// TIA Portal V17 export
// export: Created 2023-02-14T02:49:47.0513541Z, ExportSetting WithDefaults, DisplayName Totally Integrated Automation Portal, DisplayVersion V17, DisplayName TIA Portal Openness, DisplayVersion V17, DisplayName TIA Portal Teamcenter Gateway, DisplayVersion V17, DisplayName TIA Portal Version Control Interface, DisplayVersion V17, DisplayName SINAMICS Startdrive Advanced, DisplayVersion V17, DisplayName SINAMICS Startdrive G130, G150, S120, S150, SINAMICS MV, S210, DisplayVersion V17, DisplayName SINAMICS Startdrive G110M, G120, G120C, G120D, G120P, G115D, DisplayVersion V17, DisplayName STEP 7 Professional, DisplayVersion V17, DisplayName STEP 7 Safety, DisplayVersion V17, DisplayName WinCC Professional, DisplayVersion V17
FUNCTION_BLOCK "Buffer_Tank"   // FB110, LAD
{ S7_Optimized_Access := 'TRUE' }
VERSION : 0.1
// stored: AutoNumber false, IsIECCheckEnabled false, IsRetainMemResEnabled false, MemoryReserve 100, SetENOAutomatically false, UDAEnableTagReadback false
   VAR_INPUT
      IN_LT01 : Real;
      "Tank w Circulation" : Bool;
      AlarmProd_pasteur : Bool;
      HighLevel_pasteur : Bool;
      IN_FBAV_Inload : Bool;
      IN_FBAV_CIP_Tank : Bool;
      IN_FBAV_CIP_Line : Bool;
      IN_FBAV_Outlet : Bool;
      IN_FBAV_Transfer : Bool;
      IN_FBP_Transfer : Bool;
      IN_FBXA : Bool;
      IN_FBP_Circulation : Bool;
      IN_Product_Ready : Bool;
      IN_Product_TransferOnProg : Bool;
      "Inload Busy" : Bool;
      "CIP Pulse" : Bool;
      "CIP Req OK" : Bool;
      "CIP Supply ON" : Bool;
      "CIP In Progress" : Bool;
      "CIP Complete" : Bool;
      "CIP Busy" : Bool;
   END_VAR
   VAR_OUTPUT
      Out_AV_Inload : Bool;
      Out_AV_Drain_In : Bool;
      Out_AV_CIP_Tank : Bool;
      Out_AV_CIP_Line : Bool;
      Out_AV_Outlet : Bool;
      Out_AV_Transfer : Bool;
      Out_P_Transfer : Bool;
      Out_P_Transfer_SP : Real;
      Out_XA : Bool;
      Out_XA_SP : Real;
      Out_P_Circulation : Bool;
      Out_Prod_Req : Bool;
      Out_Prod_LineOpen : Bool;
      Out_CIP_Tank_Req : Bool;
      Out_CIP_Line_Req : Bool;
      Out_CIP_Tank_LineOpen : Bool;
      Out_CIP_Line_LineOpen : Bool;
   END_VAR
   VAR
      cmd : Struct
         Inload : Bool;
         Drain_In : Bool;
         Ready_for_Transfer : Bool;
         CIP_Tank : Bool;
         CIP_Line : Bool;
         Agitator_Mode : Bool;
         Agitator_Man_OnOff : Bool;
         Agitator_SpeedMode : Bool;
         Circulation : Bool;
      END_STRUCT;
   END_VAR
   VAR RETAIN
      param : Struct
         L_Lo_Lim : Real;
         L_Hi_Lim : Real := 100.0;
         L_Hys : Real := 2.0;
         "Circulation Level" : Real := 20.0;
         SP_Level_HL : Real := 100.0;
         SP_Level_ML : Real := 80.0;
         SP_Level_LL : Real := 10.0;
         DrainIn : DInt := 10;
         SP_Pump_Transfer : Real := 80.0;
         SP_Pump_CIP : Real := 80.0;
         SP_Agitator : Real := 50.0;
         SP_Level_Agi_ON1 : Real := 20.0;
         SP_Level_Agi_OFF1 : Real := 49.0;
         SP_Level_Agi_ON2 : Real := 50.0;
         SP_Level_Agi_OFF2 : Real := 64.0;
         SP_Level_Agi_ON3 : Real := 65.0;
         "CIP Ret On" : Real := 5.0;
         "CIP Ret Off" : Real;
      END_STRUCT;
   END_VAR
   VAR
      state : Struct
         "Tank LL" : Bool;
         "Tank ML" : Bool;
         "Tank HL" : Bool;
         "Tank CIP En" : Bool;
         "Tank CIP" : Bool;
         "Line CIP En" : Bool;
         "Line CIP" : Bool;
         "Ready for Transfer En" : Bool;
         "Ready for Transfer" : Bool;
         Inloading : Bool;
         "Inload En" : Bool;
         L_Agi_ON1 : Bool;
         L_Agi_ON2 : Bool;
         L_Agi_ON3 : Bool;
         Tank_Circulation : Bool;
         "Circulation Enable" : Bool;
         Circulation : Bool;
         "Transfer on Prog" : Bool;
         "CIP Return On" : Bool;
         "CIP Req" : Bool;
      END_STRUCT;
      alwaysOn : Bool;
      L_Hys_Abs : Real;
      Hys_Level_LL : Real;
      Hys_Level_ML : Real;
      Hys_Level_HL : Real;
      Hys_Level_Circ : Real;
   END_VAR
   VAR DB_SPECIFIC
      r : Struct
         PosE1 : Bool;
         PosE2 : Bool;
         PosE3 : Bool;
         PosE4 : Bool;
         PosE5 : Bool;
         PosE6 : Bool;
         PosE7 : Bool;
         PosE8 : Bool;
         PosE9 : Bool;
         PosE10 : Bool;
         PosE11 : Bool;
         PosE12 : Bool;
         PosE13 : Bool;
         PosE14 : Bool;
         PosE15 : Bool;
         PosE16 : Bool;
         PosE17 : Bool;
         PosE18 : Bool;
         PosE19 : Bool;
         PosE20 : Bool;
         PosE21 : Bool;
         PosE22 : Bool;
         PosE23 : Bool;
         PosE24 : Bool;
         PosE25 : Bool;
         PosE26 : Bool;
         PosE27 : Bool;
         PosE28 : Bool;
         PosE29 : Bool;
         PosE30 : Bool;
         PosE31 : Bool;
         PosE32 : Bool;
      END_STRUCT;
      Actuator : Struct
         AV_Inload : Bool;
         AV_Drain_In : Bool;
         AV_Outlet : Bool;
         AV_Transfer : Bool;
         AV_CIP_Tank : Bool;
         AV_CIP_Line : Bool;
         P_Transfer : Bool;
         P_CIP : Bool;
         Agitator_level : Bool;
      END_STRUCT;
   END_VAR
   VAR
      DrainIn_OnTime : TON_TIME;
      DrainIn_OffTime : TOF_TIME;
      InloadAV_OffTime : TOF_TIME;
      DrainIn_MS : DInt;
      L_AgiTim : TON_TIME;
   END_VAR
   VAR_TEMP   // added for the SCL form of the ladder/FBD networks
      _w1 : Bool;
      _w2 : Bool;
      _w3 : Bool;
   END_VAR
BEGIN

REGION Network 1: always On
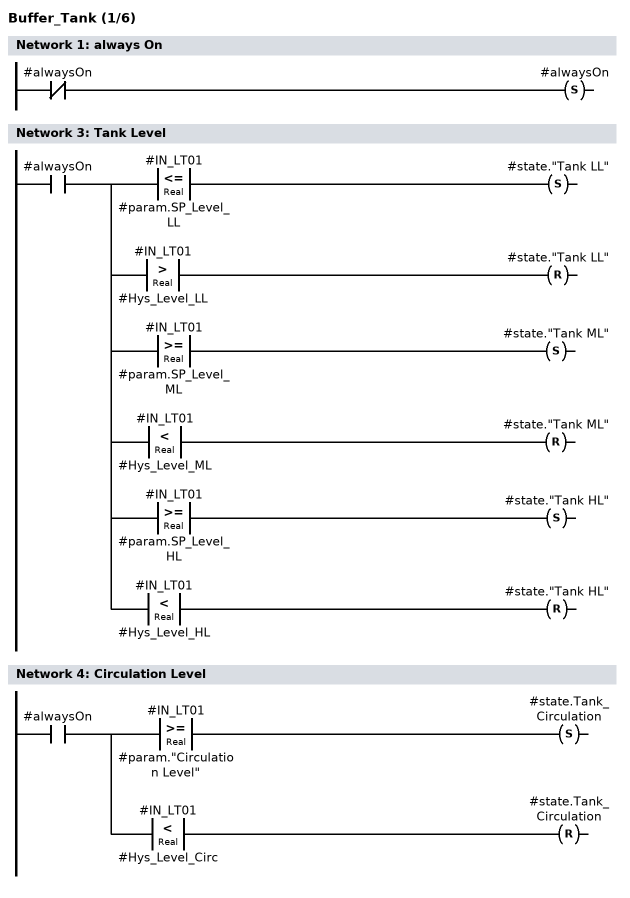
   RUNG wire#powerrail
      I_Contact( #alwaysOn )
      S_Coil( #alwaysOn )
   END_RUNG
   // the same network as SCL:
   IF NOT #alwaysOn THEN #alwaysOn := TRUE; END_IF;
END_REGION

NETWORK
TITLE = Hys Calculation
//Level Hys Absolute
      L     #param.L_Hi_Lim;
      L     #param.L_Lo_Lim;
      -R;
      L     100.0;
      /R;
      L     #param.L_Hys;
      *R;
      T     #L_Hys_Abs;
//Tank High Level
      L     #param.SP_Level_HL;
      L     #L_Hys_Abs;
      -R;
      T     #Hys_Level_HL;
//Tank Mid Level
      L     #param.SP_Level_ML;
      L     #L_Hys_Abs;
      -R;
      T     #Hys_Level_ML;
//Tank Low Level
      L     #param.SP_Level_LL;
      L     #L_Hys_Abs;
      +R;
      T     #Hys_Level_LL;
//Level Circulation
      L     #param."Circulation Level";
      L     #L_Hys_Abs;
      -R;
      T     #Hys_Level_Circ;



REGION Network 3: Tank Level
   RUNG wire#powerrail
      Contact( #alwaysOn )
      wire#w1
      { S7_Templates := "SrcType := Real" } LE_Contact(in1 := #IN_LT01, in2 := #param.SP_Level_LL)
      S_Coil( #state."Tank LL" )
   END_RUNG
   RUNG wire#w1
      { S7_Templates := "SrcType := Real" } GT_Contact(in1 := #IN_LT01, in2 := #Hys_Level_LL)
      R_Coil( #state."Tank LL" )
   END_RUNG
   RUNG wire#w1
      { S7_Templates := "SrcType := Real" } GE_Contact(in1 := #IN_LT01, in2 := #param.SP_Level_ML)
      S_Coil( #state."Tank ML" )
   END_RUNG
   RUNG wire#w1
      { S7_Templates := "SrcType := Real" } LT_Contact(in1 := #IN_LT01, in2 := #Hys_Level_ML)
      R_Coil( #state."Tank ML" )
   END_RUNG
   RUNG wire#w1
      { S7_Templates := "SrcType := Real" } GE_Contact(in1 := #IN_LT01, in2 := #param.SP_Level_HL)
      S_Coil( #state."Tank HL" )
   END_RUNG
   RUNG wire#w1
      { S7_Templates := "SrcType := Real" } LT_Contact(in1 := #IN_LT01, in2 := #Hys_Level_HL)
      R_Coil( #state."Tank HL" )
   END_RUNG
   // the same network as SCL:
   IF #alwaysOn AND (#IN_LT01 <= #param.SP_Level_LL) THEN #state."Tank LL" := TRUE; END_IF;
   IF #alwaysOn AND (#IN_LT01 > #Hys_Level_LL) THEN #state."Tank LL" := FALSE; END_IF;
   IF #alwaysOn AND (#IN_LT01 >= #param.SP_Level_ML) THEN #state."Tank ML" := TRUE; END_IF;
   IF #alwaysOn AND (#IN_LT01 < #Hys_Level_ML) THEN #state."Tank ML" := FALSE; END_IF;
   IF #alwaysOn AND (#IN_LT01 >= #param.SP_Level_HL) THEN #state."Tank HL" := TRUE; END_IF;
   IF #alwaysOn AND (#IN_LT01 < #Hys_Level_HL) THEN #state."Tank HL" := FALSE; END_IF;
END_REGION

REGION Network 4: Circulation Level
   RUNG wire#powerrail
      Contact( #alwaysOn )
      wire#w1
      { S7_Templates := "SrcType := Real" } GE_Contact(in1 := #IN_LT01, in2 := #param."Circulation Level")
      S_Coil( #state.Tank_Circulation )
   END_RUNG
   RUNG wire#w1
      { S7_Templates := "SrcType := Real" } LT_Contact(in1 := #IN_LT01, in2 := #Hys_Level_Circ)
      R_Coil( #state.Tank_Circulation )
   END_RUNG
   // the same network as SCL:
   IF #alwaysOn AND (#IN_LT01 >= #param."Circulation Level") THEN #state.Tank_Circulation := TRUE; END_IF;
   IF #alwaysOn AND (#IN_LT01 < #Hys_Level_Circ) THEN #state.Tank_Circulation := FALSE; END_IF;
END_REGION

REGION Network 5: Agitator Level ON-OFF
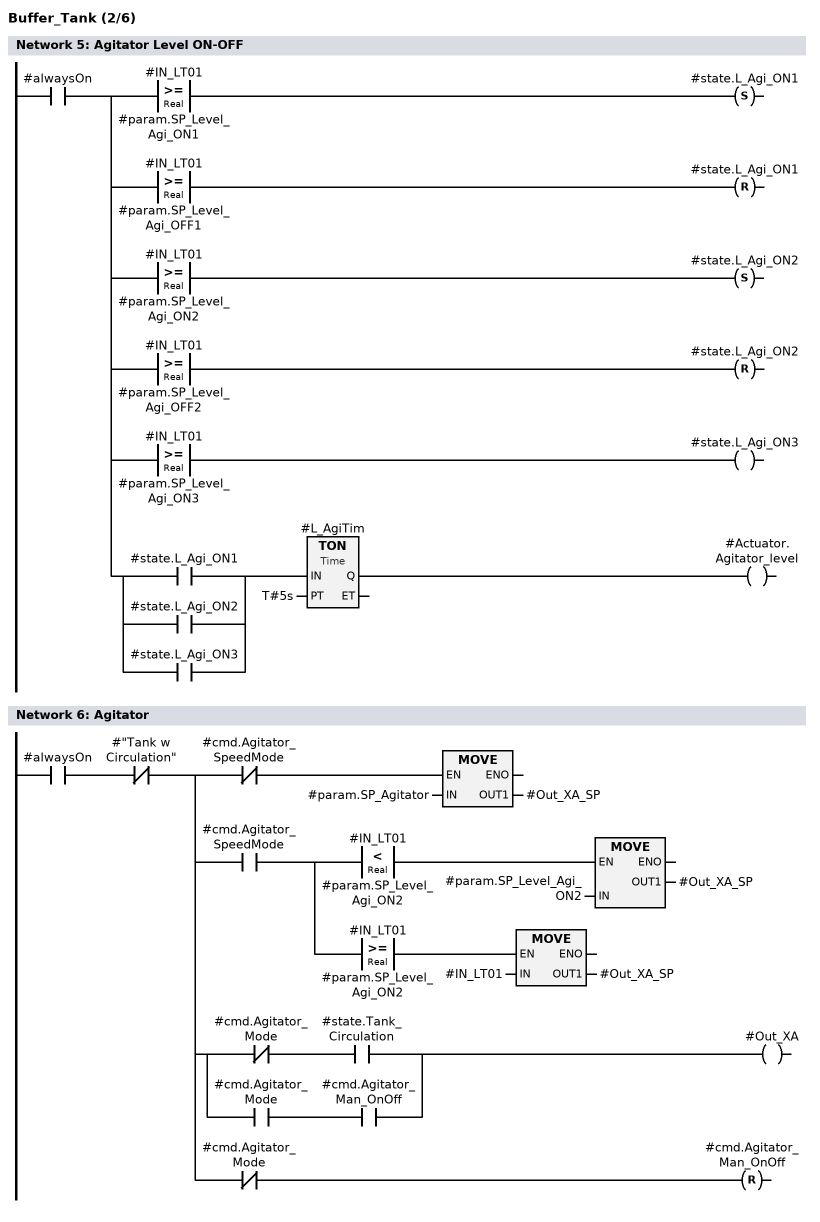
   RUNG wire#powerrail
      Contact( #alwaysOn )
      wire#w1
      { S7_Templates := "SrcType := Real" } GE_Contact(in1 := #IN_LT01, in2 := #param.SP_Level_Agi_ON1)
      S_Coil( #state.L_Agi_ON1 )
   END_RUNG
   RUNG wire#w1
      { S7_Templates := "SrcType := Real" } GE_Contact(in1 := #IN_LT01, in2 := #param.SP_Level_Agi_OFF1)
      R_Coil( #state.L_Agi_ON1 )
   END_RUNG
   RUNG wire#w1
      { S7_Templates := "SrcType := Real" } GE_Contact(in1 := #IN_LT01, in2 := #param.SP_Level_Agi_ON2)
      S_Coil( #state.L_Agi_ON2 )
   END_RUNG
   RUNG wire#w1
      { S7_Templates := "SrcType := Real" } GE_Contact(in1 := #IN_LT01, in2 := #param.SP_Level_Agi_OFF2)
      R_Coil( #state.L_Agi_ON2 )
   END_RUNG
   RUNG wire#w1
      { S7_Templates := "SrcType := Real" } GE_Contact(in1 := #IN_LT01, in2 := #param.SP_Level_Agi_ON3)
      Coil( #state.L_Agi_ON3 )
   END_RUNG
   RUNG wire#w1
      Contact( #state.L_Agi_ON1 )
      wire#w2
      { S7_Templates := "time_type := Time" } #L_AgiTim.TON(pt := T#5s, et =>)
      Coil( #Actuator.Agitator_level )
   END_RUNG
   RUNG wire#w1
      Contact( #state.L_Agi_ON2 )
   END_RUNG wire#w2
   RUNG wire#w1
      Contact( #state.L_Agi_ON3 )
   END_RUNG wire#w2
   // the same network as SCL:
   IF #alwaysOn AND (#IN_LT01 >= #param.SP_Level_Agi_ON1) THEN #state.L_Agi_ON1 := TRUE; END_IF;
   IF #alwaysOn AND (#IN_LT01 >= #param.SP_Level_Agi_OFF1) THEN #state.L_Agi_ON1 := FALSE; END_IF;
   IF #alwaysOn AND (#IN_LT01 >= #param.SP_Level_Agi_ON2) THEN #state.L_Agi_ON2 := TRUE; END_IF;
   IF #alwaysOn AND (#IN_LT01 >= #param.SP_Level_Agi_OFF2) THEN #state.L_Agi_ON2 := FALSE; END_IF;
   #state.L_Agi_ON3 := #alwaysOn AND (#IN_LT01 >= #param.SP_Level_Agi_ON3);
   #L_AgiTim(IN := #alwaysOn AND (#state.L_Agi_ON1 OR #state.L_Agi_ON2 OR #state.L_Agi_ON3), PT := T#5s);   // TON
   #Actuator.Agitator_level := #L_AgiTim.Q;
END_REGION

REGION Network 6: Agitator
   RUNG wire#powerrail
      Contact( #alwaysOn )
      I_Contact( #"Tank w Circulation" )
      wire#w1
      I_Contact( #cmd.Agitator_SpeedMode )
      Move(in := #param.SP_Agitator, out1 => #Out_XA_SP)
   END_RUNG
   RUNG wire#w1
      Contact( #cmd.Agitator_SpeedMode )
      wire#w2
      { S7_Templates := "SrcType := Real" } LT_Contact(in1 := #IN_LT01, in2 := #param.SP_Level_Agi_ON2)
      Move(in := #param.SP_Level_Agi_ON2, out1 => #Out_XA_SP)
   END_RUNG
   RUNG wire#w2
      { S7_Templates := "SrcType := Real" } GE_Contact(in1 := #IN_LT01, in2 := #param.SP_Level_Agi_ON2)
      Move(in := #IN_LT01, out1 => #Out_XA_SP)
   END_RUNG
   RUNG wire#w1
      I_Contact( #cmd.Agitator_Mode )
      Contact( #state.Tank_Circulation )
      wire#w3
      Coil( #Out_XA )
   END_RUNG
   RUNG wire#w1
      Contact( #cmd.Agitator_Mode )
      Contact( #cmd.Agitator_Man_OnOff )
   END_RUNG wire#w3
   RUNG wire#w1
      I_Contact( #cmd.Agitator_Mode )
      R_Coil( #cmd.Agitator_Man_OnOff )
   END_RUNG
   // the same network as SCL:
   #_w1 := #alwaysOn AND NOT #"Tank w Circulation";
   IF #_w1 AND NOT #cmd.Agitator_SpeedMode THEN #Out_XA_SP := #param.SP_Agitator; END_IF;
   #_w2 := #_w1 AND #cmd.Agitator_SpeedMode;
   IF #_w2 AND (#IN_LT01 < #param.SP_Level_Agi_ON2) THEN #Out_XA_SP := #param.SP_Level_Agi_ON2; END_IF;
   IF #_w2 AND (#IN_LT01 >= #param.SP_Level_Agi_ON2) THEN #Out_XA_SP := #IN_LT01; END_IF;
   #Out_XA := #_w1 AND ((NOT #cmd.Agitator_Mode AND #state.Tank_Circulation) OR (#cmd.Agitator_Mode AND #cmd.Agitator_Man_OnOff));
   IF #_w1 AND NOT #cmd.Agitator_Mode THEN #cmd.Agitator_Man_OnOff := FALSE; END_IF;
END_REGION

REGION Network 7: Circulation
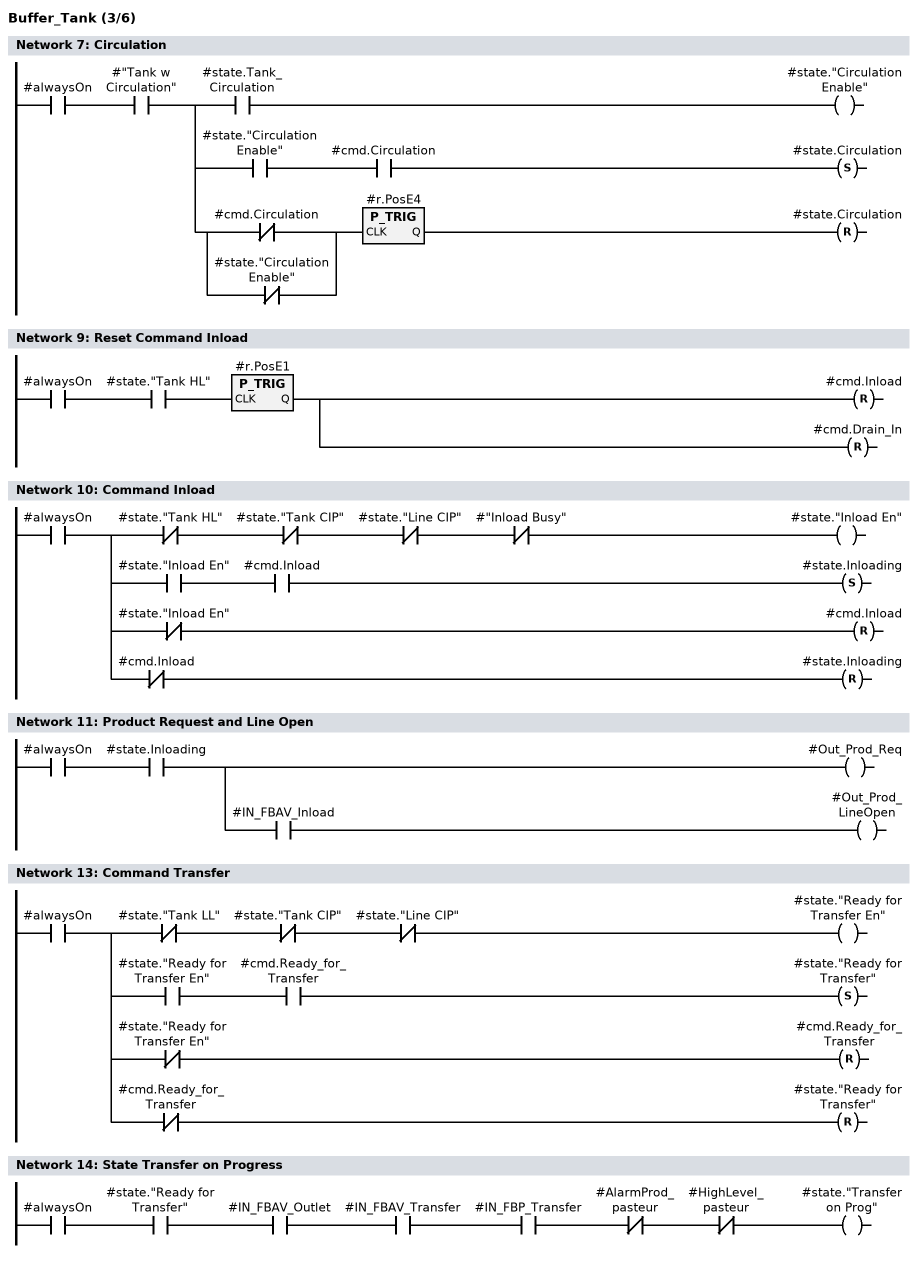
   RUNG wire#powerrail
      Contact( #alwaysOn )
      Contact( #"Tank w Circulation" )
      wire#w1
      Contact( #state.Tank_Circulation )
      Coil( #state."Circulation Enable" )
   END_RUNG
   RUNG wire#w1
      Contact( #state."Circulation Enable" )
      Contact( #cmd.Circulation )
      S_Coil( #state.Circulation )
   END_RUNG
   RUNG wire#w1
      I_Contact( #cmd.Circulation )
      wire#w2
      P_Trig( #r.PosE4 )
      R_Coil( #state.Circulation )
   END_RUNG
   RUNG wire#w1
      I_Contact( #state."Circulation Enable" )
   END_RUNG wire#w2
   // the same network as SCL:
   #_w1 := #alwaysOn AND #"Tank w Circulation";
   #state."Circulation Enable" := #_w1 AND #state.Tank_Circulation;
   IF #_w1 AND #state."Circulation Enable" AND #cmd.Circulation THEN #state.Circulation := TRUE; END_IF;
   #_w2 := #_w1 AND (NOT #cmd.Circulation OR NOT #state."Circulation Enable");
   #_w3 := #_w2 AND NOT #r.PosE4;   // rising edge
   #r.PosE4 := #_w2;
   IF #_w3 THEN #state.Circulation := FALSE; END_IF;
END_REGION

REGION Network 9: Reset Command Inload
   RUNG wire#powerrail
      Contact( #alwaysOn )
      Contact( #state."Tank HL" )
      P_Trig( #r.PosE1 )
      wire#w1
      R_Coil( #cmd.Inload )
   END_RUNG
   RUNG wire#w1
      R_Coil( #cmd.Drain_In )
   END_RUNG
   // the same network as SCL:
   #_w1 := #alwaysOn AND #state."Tank HL";
   #_w2 := #_w1 AND NOT #r.PosE1;   // rising edge
   #r.PosE1 := #_w1;
   IF #_w2 THEN
       #cmd.Inload := FALSE;
       #cmd.Drain_In := FALSE;
   END_IF;
END_REGION

REGION Network 10: Command Inload
   RUNG wire#powerrail
      Contact( #alwaysOn )
      wire#w1
      I_Contact( #state."Tank HL" )
      I_Contact( #state."Tank CIP" )
      I_Contact( #state."Line CIP" )
      I_Contact( #"Inload Busy" )
      Coil( #state."Inload En" )
   END_RUNG
   RUNG wire#w1
      Contact( #state."Inload En" )
      Contact( #cmd.Inload )
      S_Coil( #state.Inloading )
   END_RUNG
   RUNG wire#w1
      I_Contact( #state."Inload En" )
      R_Coil( #cmd.Inload )
   END_RUNG
   RUNG wire#w1
      I_Contact( #cmd.Inload )
      R_Coil( #state.Inloading )
   END_RUNG
   // the same network as SCL:
   #state."Inload En" := #alwaysOn AND NOT #state."Tank HL" AND NOT #state."Tank CIP" AND NOT #state."Line CIP" AND NOT #"Inload Busy";
   IF #alwaysOn AND #state."Inload En" AND #cmd.Inload THEN #state.Inloading := TRUE; END_IF;
   IF #alwaysOn AND NOT #state."Inload En" THEN #cmd.Inload := FALSE; END_IF;
   IF #alwaysOn AND NOT #cmd.Inload THEN #state.Inloading := FALSE; END_IF;
END_REGION

REGION Network 11: Product Request and Line Open
   RUNG wire#powerrail
      Contact( #alwaysOn )
      Contact( #state.Inloading )
      wire#w1
      Coil( #Out_Prod_Req )
   END_RUNG
   RUNG wire#w1
      Contact( #IN_FBAV_Inload )
      Coil( #Out_Prod_LineOpen )
   END_RUNG
   // the same network as SCL:
   #Out_Prod_Req := #alwaysOn AND #state.Inloading;
   #Out_Prod_LineOpen := #Out_Prod_Req AND #IN_FBAV_Inload;
END_REGION

REGION Network 13: Command Transfer
   RUNG wire#powerrail
      Contact( #alwaysOn )
      wire#w1
      I_Contact( #state."Tank LL" )
      I_Contact( #state."Tank CIP" )
      I_Contact( #state."Line CIP" )
      Coil( #state."Ready for Transfer En" )
   END_RUNG
   RUNG wire#w1
      Contact( #state."Ready for Transfer En" )
      Contact( #cmd.Ready_for_Transfer )
      S_Coil( #state."Ready for Transfer" )
   END_RUNG
   RUNG wire#w1
      I_Contact( #state."Ready for Transfer En" )
      R_Coil( #cmd.Ready_for_Transfer )
   END_RUNG
   RUNG wire#w1
      I_Contact( #cmd.Ready_for_Transfer )
      R_Coil( #state."Ready for Transfer" )
   END_RUNG
   // the same network as SCL:
   #state."Ready for Transfer En" := #alwaysOn AND NOT #state."Tank LL" AND NOT #state."Tank CIP" AND NOT #state."Line CIP";
   IF #alwaysOn AND #state."Ready for Transfer En" AND #cmd.Ready_for_Transfer THEN
       #state."Ready for Transfer" := TRUE;
   END_IF;
   IF #alwaysOn AND NOT #state."Ready for Transfer En" THEN #cmd.Ready_for_Transfer := FALSE; END_IF;
   IF #alwaysOn AND NOT #cmd.Ready_for_Transfer THEN #state."Ready for Transfer" := FALSE; END_IF;
END_REGION

REGION Network 14: State Transfer on Progress
   RUNG wire#powerrail
      Contact( #alwaysOn )
      Contact( #state."Ready for Transfer" )
      Contact( #IN_FBAV_Outlet )
      Contact( #IN_FBAV_Transfer )
      Contact( #IN_FBP_Transfer )
      I_Contact( #AlarmProd_pasteur )
      I_Contact( #HighLevel_pasteur )
      Coil( #state."Transfer on Prog" )
   END_RUNG
   // the same network as SCL:
   #state."Transfer on Prog" := #alwaysOn AND #state."Ready for Transfer" AND #IN_FBAV_Outlet AND #IN_FBAV_Transfer AND #IN_FBP_Transfer AND NOT #AlarmProd_pasteur AND NOT #HighLevel_pasteur;
END_REGION

REGION Network 16: Command CIP
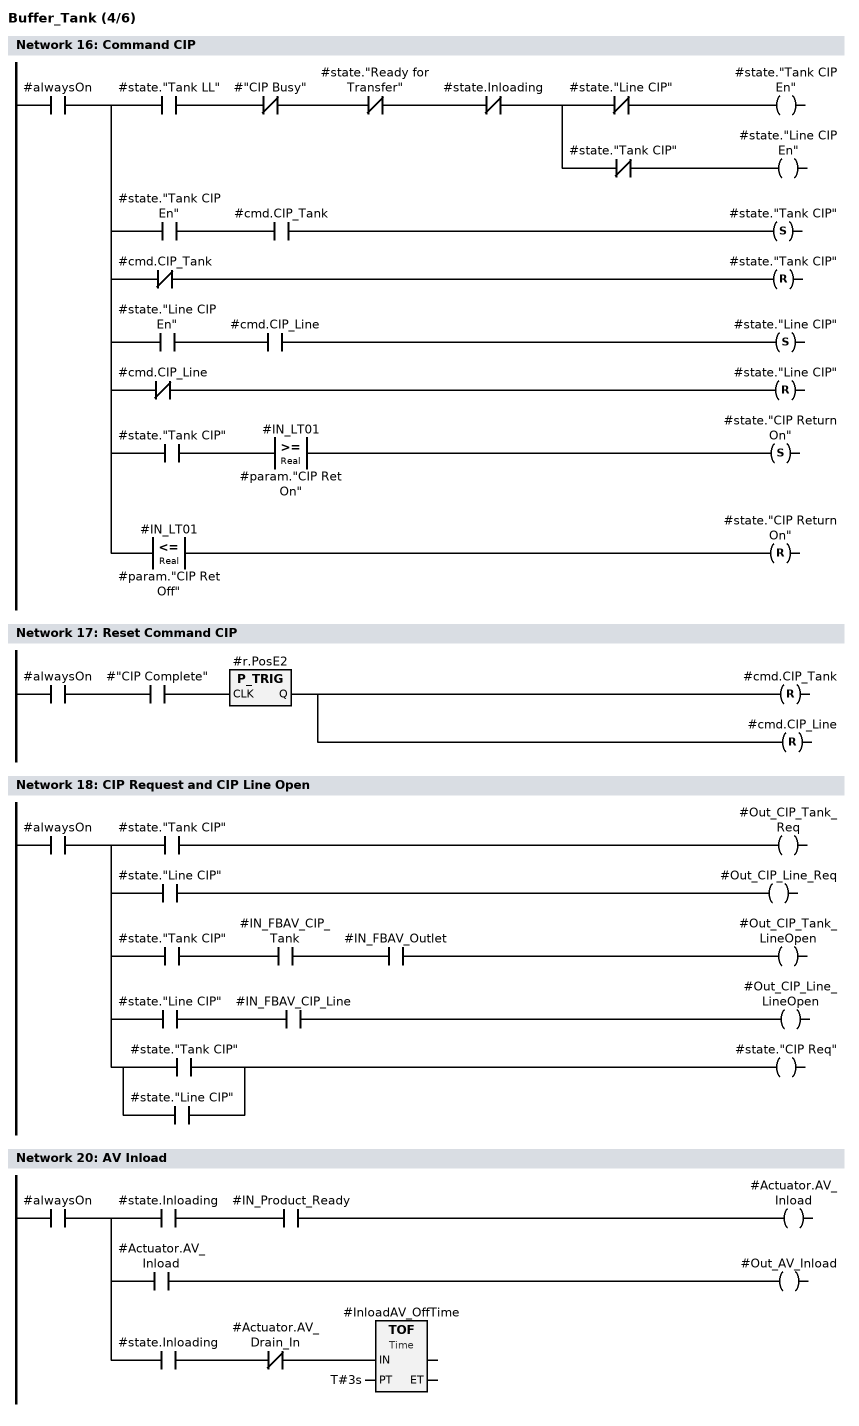
   RUNG wire#powerrail
      Contact( #alwaysOn )
      wire#w1
      Contact( #state."Tank LL" )
      I_Contact( #"CIP Busy" )
      I_Contact( #state."Ready for Transfer" )
      I_Contact( #state.Inloading )
      wire#w2
      I_Contact( #state."Line CIP" )
      Coil( #state."Tank CIP En" )
   END_RUNG
   RUNG wire#w2
      I_Contact( #state."Tank CIP" )
      Coil( #state."Line CIP En" )
   END_RUNG
   RUNG wire#w1
      Contact( #state."Tank CIP En" )
      Contact( #cmd.CIP_Tank )
      S_Coil( #state."Tank CIP" )
   END_RUNG
   RUNG wire#w1
      I_Contact( #cmd.CIP_Tank )
      R_Coil( #state."Tank CIP" )
   END_RUNG
   RUNG wire#w1
      Contact( #state."Line CIP En" )
      Contact( #cmd.CIP_Line )
      S_Coil( #state."Line CIP" )
   END_RUNG
   RUNG wire#w1
      I_Contact( #cmd.CIP_Line )
      R_Coil( #state."Line CIP" )
   END_RUNG
   RUNG wire#w1
      Contact( #state."Tank CIP" )
      { S7_Templates := "SrcType := Real" } GE_Contact(in1 := #IN_LT01, in2 := #param."CIP Ret On")
      S_Coil( #state."CIP Return On" )
   END_RUNG
   RUNG wire#w1
      { S7_Templates := "SrcType := Real" } LE_Contact(in1 := #IN_LT01, in2 := #param."CIP Ret Off")
      R_Coil( #state."CIP Return On" )
   END_RUNG
   // the same network as SCL:
   #_w1 := #alwaysOn AND #state."Tank LL" AND NOT #"CIP Busy" AND NOT #state."Ready for Transfer" AND NOT #state.Inloading;
   #state."Tank CIP En" := #_w1 AND NOT #state."Line CIP";
   #state."Line CIP En" := #_w1 AND NOT #state."Tank CIP";
   IF #alwaysOn AND #state."Tank CIP En" AND #cmd.CIP_Tank THEN #state."Tank CIP" := TRUE; END_IF;
   IF #alwaysOn AND NOT #cmd.CIP_Tank THEN #state."Tank CIP" := FALSE; END_IF;
   IF #alwaysOn AND #state."Line CIP En" AND #cmd.CIP_Line THEN #state."Line CIP" := TRUE; END_IF;
   IF #alwaysOn AND NOT #cmd.CIP_Line THEN #state."Line CIP" := FALSE; END_IF;
   IF #alwaysOn AND #state."Tank CIP" AND (#IN_LT01 >= #param."CIP Ret On") THEN
       #state."CIP Return On" := TRUE;
   END_IF;
   IF #alwaysOn AND (#IN_LT01 <= #param."CIP Ret Off") THEN #state."CIP Return On" := FALSE; END_IF;
END_REGION

REGION Network 17: Reset Command CIP
   RUNG wire#powerrail
      Contact( #alwaysOn )
      Contact( #"CIP Complete" )
      P_Trig( #r.PosE2 )
      wire#w1
      R_Coil( #cmd.CIP_Tank )
   END_RUNG
   RUNG wire#w1
      R_Coil( #cmd.CIP_Line )
   END_RUNG
   // the same network as SCL:
   #_w1 := #alwaysOn AND #"CIP Complete";
   #_w2 := #_w1 AND NOT #r.PosE2;   // rising edge
   #r.PosE2 := #_w1;
   IF #_w2 THEN
       #cmd.CIP_Tank := FALSE;
       #cmd.CIP_Line := FALSE;
   END_IF;
END_REGION

REGION Network 18: CIP Request and CIP Line Open
   RUNG wire#powerrail
      Contact( #alwaysOn )
      wire#w1
      Contact( #state."Tank CIP" )
      Coil( #Out_CIP_Tank_Req )
   END_RUNG
   RUNG wire#w1
      Contact( #state."Line CIP" )
      Coil( #Out_CIP_Line_Req )
   END_RUNG
   RUNG wire#w1
      Contact( #state."Tank CIP" )
      Contact( #IN_FBAV_CIP_Tank )
      Contact( #IN_FBAV_Outlet )
      Coil( #Out_CIP_Tank_LineOpen )
   END_RUNG
   RUNG wire#w1
      Contact( #state."Line CIP" )
      Contact( #IN_FBAV_CIP_Line )
      Coil( #Out_CIP_Line_LineOpen )
   END_RUNG
   RUNG wire#w1
      Contact( #state."Tank CIP" )
      wire#w2
      Coil( #state."CIP Req" )
   END_RUNG
   RUNG wire#w1
      Contact( #state."Line CIP" )
   END_RUNG wire#w2
   // the same network as SCL:
   #Out_CIP_Tank_Req := #alwaysOn AND #state."Tank CIP";
   #Out_CIP_Line_Req := #alwaysOn AND #state."Line CIP";
   #Out_CIP_Tank_LineOpen := #alwaysOn AND #state."Tank CIP" AND #IN_FBAV_CIP_Tank AND #IN_FBAV_Outlet;
   #Out_CIP_Line_LineOpen := #alwaysOn AND #state."Line CIP" AND #IN_FBAV_CIP_Line;
   #state."CIP Req" := #alwaysOn AND (#state."Tank CIP" OR #state."Line CIP");
END_REGION

REGION Network 20: AV Inload
   RUNG wire#powerrail
      Contact( #alwaysOn )
      wire#w1
      Contact( #state.Inloading )
      Contact( #IN_Product_Ready )
      Coil( #Actuator.AV_Inload )
   END_RUNG
   RUNG wire#w1
      Contact( #Actuator.AV_Inload )
      Coil( #Out_AV_Inload )
   END_RUNG
   RUNG wire#w1
      Contact( #state.Inloading )
      I_Contact( #Actuator.AV_Drain_In )
      { S7_Templates := "time_type := Time" } #InloadAV_OffTime.TOF(pt := T#3s, et =>)
   END_RUNG
   // the same network as SCL:
   #Actuator.AV_Inload := #alwaysOn AND #state.Inloading AND #IN_Product_Ready;
   #Out_AV_Inload := #alwaysOn AND #Actuator.AV_Inload;
   #InloadAV_OffTime(IN := #alwaysOn AND #state.Inloading AND NOT #Actuator.AV_Drain_In, PT := T#3s);   // TOF
END_REGION

REGION Network 21: AV Drain In
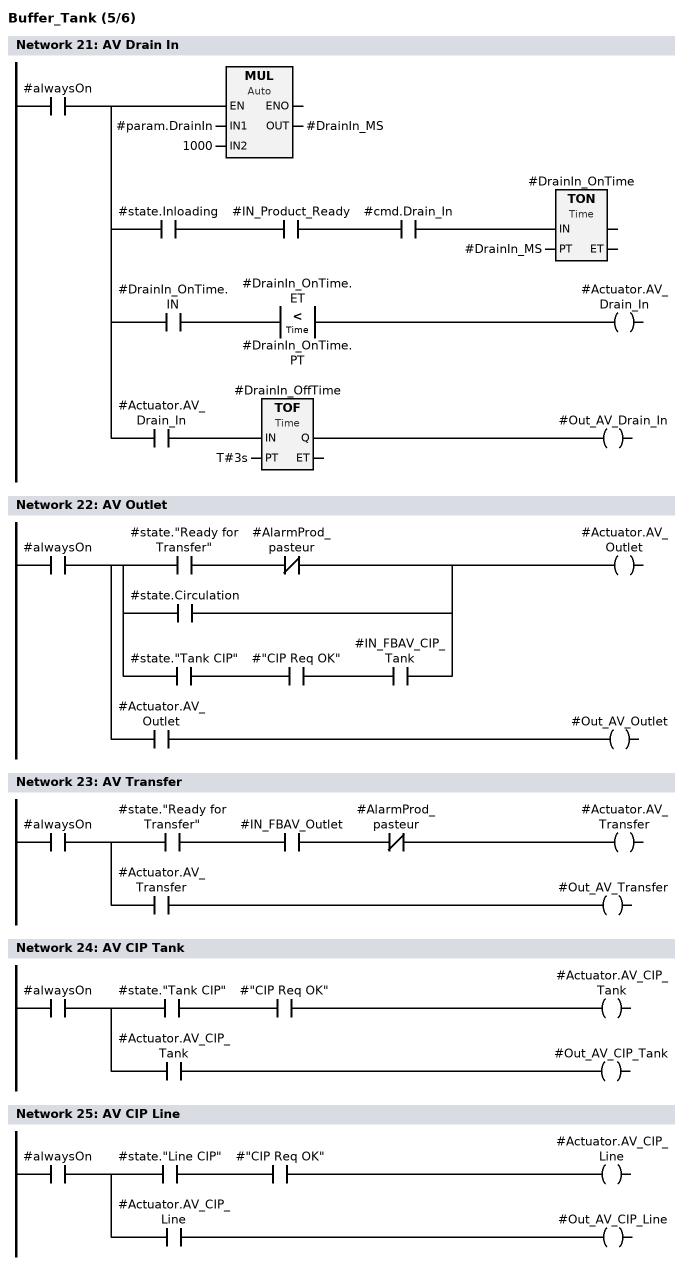
   RUNG wire#powerrail
      Contact( #alwaysOn )
      wire#w1
      Mul(in1 := #param.DrainIn, in2 := 1000, out => #DrainIn_MS)
   END_RUNG
   RUNG wire#w1
      Contact( #state.Inloading )
      Contact( #IN_Product_Ready )
      Contact( #cmd.Drain_In )
      { S7_Templates := "time_type := Time" } #DrainIn_OnTime.TON(pt := #DrainIn_MS, et =>)
   END_RUNG
   RUNG wire#w1
      Contact( #DrainIn_OnTime.IN )
      { S7_Templates := "SrcType := Time" } LT_Contact(in1 := #DrainIn_OnTime.ET, in2 := #DrainIn_OnTime.PT)
      Coil( #Actuator.AV_Drain_In )
   END_RUNG
   RUNG wire#w1
      Contact( #Actuator.AV_Drain_In )
      { S7_Templates := "time_type := Time" } #DrainIn_OffTime.TOF(pt := T#3s, et =>)
      Coil( #Out_AV_Drain_In )
   END_RUNG
   // the same network as SCL:
   IF #alwaysOn THEN #DrainIn_MS := #param.DrainIn * 1000; END_IF;
   #DrainIn_OnTime(IN := #alwaysOn AND #state.Inloading AND #IN_Product_Ready AND #cmd.Drain_In,   // TON
                   PT := #DrainIn_MS);
   #Actuator.AV_Drain_In := #alwaysOn AND #DrainIn_OnTime.IN AND (#DrainIn_OnTime.ET < #DrainIn_OnTime.PT);
   #DrainIn_OffTime(IN := #alwaysOn AND #Actuator.AV_Drain_In, PT := T#3s);   // TOF
   #Out_AV_Drain_In := #DrainIn_OffTime.Q;
END_REGION

REGION Network 22: AV Outlet
   RUNG wire#powerrail
      Contact( #alwaysOn )
      wire#w1
      Contact( #state."Ready for Transfer" )
      I_Contact( #AlarmProd_pasteur )
      wire#w2
      Coil( #Actuator.AV_Outlet )
   END_RUNG
   RUNG wire#w1
      Contact( #state.Circulation )
   END_RUNG wire#w2
   RUNG wire#w1
      Contact( #state."Tank CIP" )
      Contact( #"CIP Req OK" )
      Contact( #IN_FBAV_CIP_Tank )
   END_RUNG wire#w2
   RUNG wire#w1
      Contact( #Actuator.AV_Outlet )
      Coil( #Out_AV_Outlet )
   END_RUNG
   // the same network as SCL:
   #Actuator.AV_Outlet := #alwaysOn AND ((#state."Ready for Transfer" AND NOT #AlarmProd_pasteur) OR #state.Circulation OR (#state."Tank CIP" AND #"CIP Req OK" AND #IN_FBAV_CIP_Tank));
   #Out_AV_Outlet := #alwaysOn AND #Actuator.AV_Outlet;
END_REGION

REGION Network 23: AV Transfer
   RUNG wire#powerrail
      Contact( #alwaysOn )
      wire#w1
      Contact( #state."Ready for Transfer" )
      Contact( #IN_FBAV_Outlet )
      I_Contact( #AlarmProd_pasteur )
      Coil( #Actuator.AV_Transfer )
   END_RUNG
   RUNG wire#w1
      Contact( #Actuator.AV_Transfer )
      Coil( #Out_AV_Transfer )
   END_RUNG
   // the same network as SCL:
   #Actuator.AV_Transfer := #alwaysOn AND #state."Ready for Transfer" AND #IN_FBAV_Outlet AND NOT #AlarmProd_pasteur;
   #Out_AV_Transfer := #alwaysOn AND #Actuator.AV_Transfer;
END_REGION

REGION Network 24: AV CIP Tank
   RUNG wire#powerrail
      Contact( #alwaysOn )
      wire#w1
      Contact( #state."Tank CIP" )
      Contact( #"CIP Req OK" )
      Coil( #Actuator.AV_CIP_Tank )
   END_RUNG
   RUNG wire#w1
      Contact( #Actuator.AV_CIP_Tank )
      Coil( #Out_AV_CIP_Tank )
   END_RUNG
   // the same network as SCL:
   #Actuator.AV_CIP_Tank := #alwaysOn AND #state."Tank CIP" AND #"CIP Req OK";
   #Out_AV_CIP_Tank := #alwaysOn AND #Actuator.AV_CIP_Tank;
END_REGION

REGION Network 25: AV CIP Line
   RUNG wire#powerrail
      Contact( #alwaysOn )
      wire#w1
      Contact( #state."Line CIP" )
      Contact( #"CIP Req OK" )
      Coil( #Actuator.AV_CIP_Line )
   END_RUNG
   RUNG wire#w1
      Contact( #Actuator.AV_CIP_Line )
      Coil( #Out_AV_CIP_Line )
   END_RUNG
   // the same network as SCL:
   #Actuator.AV_CIP_Line := #alwaysOn AND #state."Line CIP" AND #"CIP Req OK";
   #Out_AV_CIP_Line := #alwaysOn AND #Actuator.AV_CIP_Line;
END_REGION

REGION Network 27: Pump Transfer
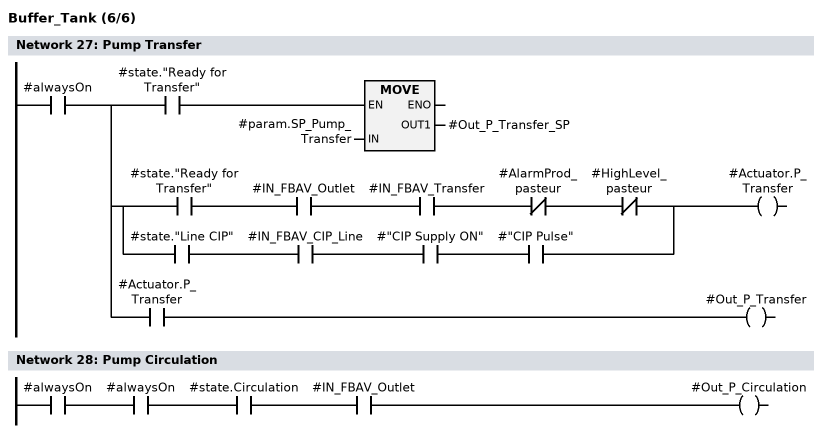
   RUNG wire#powerrail
      Contact( #alwaysOn )
      wire#w1
      Contact( #state."Ready for Transfer" )
      Move(in := #param.SP_Pump_Transfer, out1 => #Out_P_Transfer_SP)
   END_RUNG
   RUNG wire#w1
      Contact( #state."Ready for Transfer" )
      Contact( #IN_FBAV_Outlet )
      Contact( #IN_FBAV_Transfer )
      I_Contact( #AlarmProd_pasteur )
      I_Contact( #HighLevel_pasteur )
      wire#w2
      Coil( #Actuator.P_Transfer )
   END_RUNG
   RUNG wire#w1
      Contact( #state."Line CIP" )
      Contact( #IN_FBAV_CIP_Line )
      Contact( #"CIP Supply ON" )
      Contact( #"CIP Pulse" )
   END_RUNG wire#w2
   RUNG wire#w1
      Contact( #Actuator.P_Transfer )
      Coil( #Out_P_Transfer )
   END_RUNG
   // the same network as SCL:
   IF #alwaysOn AND #state."Ready for Transfer" THEN #Out_P_Transfer_SP := #param.SP_Pump_Transfer; END_IF;
   #Actuator.P_Transfer := #alwaysOn AND ((#state."Ready for Transfer" AND #IN_FBAV_Outlet AND #IN_FBAV_Transfer AND NOT #AlarmProd_pasteur AND NOT #HighLevel_pasteur) OR (#state."Line CIP" AND #IN_FBAV_CIP_Line AND #"CIP Supply ON" AND #"CIP Pulse"));
   #Out_P_Transfer := #alwaysOn AND #Actuator.P_Transfer;
END_REGION

REGION Network 28: Pump Circulation
   RUNG wire#powerrail
      Contact( #alwaysOn )
      Contact( #alwaysOn )
      Contact( #state.Circulation )
      Contact( #IN_FBAV_Outlet )
      Coil( #Out_P_Circulation )
   END_RUNG
   // the same network as SCL:
   #Out_P_Circulation := #alwaysOn AND #alwaysOn AND #state.Circulation AND #IN_FBAV_Outlet;
END_REGION
END_FUNCTION_BLOCK
